// TIA Portal V18 export
// export: Created 2025-12-01T12:39:34.8419056Z, ExportSetting None, DisplayName Totally Integrated Automation Portal, DisplayVersion V18 Update 5, DisplayName TIA Portal Openness, DisplayVersion V18 Update 5, DisplayName TIA Portal Teamcenter Gateway, DisplayVersion V18, DisplayName TIA Portal Version Control Interface, DisplayVersion V18, DisplayName STEP 7 Professional, DisplayVersion V18 Update 5, DisplayName STEP 7 Safety, DisplayVersion V18, DisplayName WinCC Professional, DisplayVersion V18 Update 5
VAR_GLOBAL   // PLC tag table "PLCIO_DQ"
   oHMIControlOn AT %Q100.0 : Bool;   // HMI_上电按钮
   oHMIMachineStart AT %Q100.1 : Bool;   // HMI_设备启动按钮
   oHMIMachineStop AT %Q100.2 : Bool;   // HMI_设备停止按钮
   oHMIResetButton AT %Q100.3 : Bool;   // HMI_复位按钮
   oHMISafetyGateUnlock AT %Q100.4 : Bool;   // HMI_安全门解锁按钮
   "RESERVE_Q100.5" AT %Q100.5 : Bool;   // 备用_Q100.5
   "RESERVE_Q100.6" AT %Q100.6 : Bool;   // 备用_Q100.6
   "RESERVE_Q100.7" AT %Q100.7 : Bool;   // 备用_Q100.7
   "oTowerLight-Green" AT %Q101.0 : Bool;   // 稳光-绿
   "oTowerLight-Red" AT %Q101.1 : Bool;   // 稳光-红
   "oTowerLight-yellow" AT %Q101.2 : Bool;   // 稳光-黄
   "oTowerLight-Blue" AT %Q101.3 : Bool;   // 稳光-蓝
   "oTowerLight-Buzzer" AT %Q101.4 : Bool;   // 蜂鸣
   oLED_lamp_1 AT %Q101.5 : Bool;   // 日光灯_1
   oLED_lamp_2 AT %Q101.6 : Bool;   // 日光灯_2
   oSafetyPLC AT %Q101.7 : Bool;   // 安全PLC
   oSafetyDoorLocked_1 AT %Q102.0 : Bool;   // 安全门锁定_1
   oSafetyDoorLocked_2 AT %Q102.1 : Bool;   // 安全门锁定_2
   oSafetyDoorLocked_3 AT %Q102.2 : Bool;   // 安全门锁定_3
   oSafetyDoorLocked_4 AT %Q102.3 : Bool;   // 安全门锁定_4
   oSafetyDoorLocked_5 AT %Q102.4 : Bool;   // 安全门锁定_5
   oSafetyDoorLocked_6 AT %Q102.5 : Bool;   // 安全门锁定_6
   oSafetyDoorLocked_7 AT %Q102.6 : Bool;   // 安全门锁定_7
   oSafetyDoorLocked_8 AT %Q102.7 : Bool;   // 安全门锁定_8
   oSafetyDoorLocked AT %Q103.0 : Bool;   // 连锁安全门锁定
   "oE-NG-01SafetyGate" AT %Q103.1 : Bool;   // E-NG料盒-01安全门锁
   oMaterielDoorLocked_H2 AT %Q103.4 : Bool;   // 物料门锁定_2
   oMaterielDoorLocked_J1 AT %Q103.5 : Bool;   // 物料门锁定_3
   "oE-NG-02SafetyGate" AT %Q103.2 : Bool;   // E-NG料盒-02安全门锁
   oMaterielDoorLocked_H1 AT %Q103.3 : Bool;   // 物料门锁定_1
   oMaterielDoorLocked_J2 AT %Q103.6 : Bool;   // 物料门锁定_4
   oMaterielDoorLocked_K1 AT %Q103.7 : Bool;   // 物料门锁定_5
   oNG_Button1 AT %Q104.0 : Bool;   // NG下料按钮1
   oNG_Button2 AT %Q104.1 : Bool;   // NG下料按钮2
   oShaft_Button AT %Q104.2 : Bool;   // shaft 上料按钮
   oShaft_EmptyButton AT %Q104.3 : Bool;   // shaft 取空料盘按钮
   oMagnet_Button AT %Q104.4 : Bool;   // Magnet上料按钮
   oMagnet_EmptyButton AT %Q104.5 : Bool;   // Magnet取空料盘按钮
   oMagnet_UnlockButton AT %Q104.6 : Bool;   // Magne门解锁按钮
   "RESERVE_Q104.7" AT %Q104.7 : Bool;   // 备用_Q104.7
   oUnloading_EmptyButton AT %Q105.4 : Bool;   // Unloading取空料盘按钮
   oUnloading_UnlockButton AT %Q105.5 : Bool;   // Unloading门解锁按钮
   oMaterielDoorLocked_K2 AT %Q105.6 : Bool;   // 物料门锁定_6
   oMaterielDoorLocked_L1 AT %Q105.7 : Bool;   // 物料门锁定_7
   oReserved_Button AT %Q105.0 : Bool;   // Reserved上料按钮
   oReserved_EmptyButton AT %Q105.1 : Bool;   // Reserved取空料盘按钮
   oReserved_UnlockButton AT %Q105.2 : Bool;   // Reserved门解锁按钮
   oUnloading_Button AT %Q105.3 : Bool;   // Unloading按钮
   "oC-GluingPro_X" AT %Q106.0 : Bool;   // C-涂胶模组点胶阀_a / C-涂胶系统程序X
   "oC-GluingPro_Y" AT %Q106.1 : Bool;   // C-涂胶模组点胶阀_b / C-涂胶系统程序Y
   "oC-GluingReset" AT %Q106.2 : Bool;   // C-涂胶模组点胶阀_c / C-涂胶系统复位
   "oC-GluingPro_Z" AT %Q106.3 : Bool;   // 备用_Q106.3 / C-涂胶系统程序Z
   "oH-shaftLifting_SpeedChange" AT %Q106.4 : Bool;   // H-shaft 顶升位驱动电机_速度切换
   "oH-shaftLifting_Start" AT %Q106.5 : Bool;   // H-shaft 顶升位驱动电机_启动进料
   "oJ-magnetLifting_SpeedChange" AT %Q106.6 : Bool;   // J-magnet顶升驱动电机_速度切换
   "oJ-magnetLifting_Start" AT %Q106.7 : Bool;   // J-magnet顶升驱动电机_启动进料
   "oK-Lifting3_SpeedChange" AT %Q107.0 : Bool;   // K-预留顶升位3驱动电机_速度切换
   "oK-Lifting3_Start" AT %Q107.1 : Bool;   // K-预留顶升位3驱动电机_启动进料
   "oL-Unloading_CCW" AT %Q107.2 : Bool;   // L-下料线体移栽电机_出料
   "oL-Unloading_CW" AT %Q107.3 : Bool;   // L-下料线体移栽电机_进料
   "oH-shaftLifting_CCWStart" AT %Q107.4 : Bool;   // H-shaft 顶升位驱动电机_启动反转出料
   "oJ-magnetLifting_CCWStart" AT %Q107.5 : Bool;   // J-magnet顶升驱动电机_启动反转出料
   "oK-Lifting3_CCWStart" AT %Q107.6 : Bool;   // K-预留顶升位3驱动电机_启动反转出料
   "RESERVE_Q107.7" AT %Q107.7 : Bool;   // 备用_Q107.7
   "oH-shaftLoading_CCW" AT %Q108.0 : Bool;   // H-shaft上料线体驱动电机_反转
   "oH-shaftLoading_CW" AT %Q108.1 : Bool;   // H-shaft上料线体驱动电机_正转
   "oH-shaftTake_CW" AT %Q108.2 : Bool;   // H-shaft取空盘驱动电机_正转
   "oH-shaftTake_CCW" AT %Q108.3 : Bool;   // H-shaft取空盘驱动电机_反转
   "RESERVE_Q108.4" AT %Q108.4 : Bool;   // 备用_Q108.4
   "RESERVE_Q108.5" AT %Q108.5 : Bool;   // 备用_Q108.5
   "RESERVE_Q108.6" AT %Q108.6 : Bool;   // 备用_Q108.6
   "RESERVE_Q108.7" AT %Q108.7 : Bool;   // 备用_Q108.7
   "RESERVE_Q109.0" AT %Q109.0 : Bool;
   "RESERVE_Q109.1" AT %Q109.1 : Bool;
   "RESERVE_Q109.2" AT %Q109.2 : Bool;
   "RESERVE_Q109.3" AT %Q109.3 : Bool;
   "RESERVE_Q109.4" AT %Q109.4 : Bool;
   "RESERVE_Q109.5" AT %Q109.5 : Bool;
   "RESERVE_Q109.6" AT %Q109.6 : Bool;
   "RESERVE_Q109.7" AT %Q109.7 : Bool;
   "J-magnet Loading _CCW" AT %Q110.0 : Bool;   // J-magnet上料线体驱动电机_反转
   "J-magnet Loading _CW" AT %Q110.1 : Bool;   // J-magnet上料线体驱动电机_正转
   "J-magnet Take _CW" AT %Q110.2 : Bool;   // J-magnet取空盘驱动电机_正转
   "J-magnet Take _CCW" AT %Q110.3 : Bool;   // J-magnet取空盘驱动电机_反转
   "RESERVE_Q110.4" AT %Q110.4 : Bool;   // 备用_Q110.4
   "RESERVE_Q110.5" AT %Q110.5 : Bool;   // 备用_Q110.5
   "RESERVE_Q110.6" AT %Q110.6 : Bool;   // 备用_Q110.6
   "RESERVE_Q110.7" AT %Q110.7 : Bool;   // 备用_Q110.7
   "RESERVE_Q111.0" AT %Q111.0 : Bool;
   "RESERVE_Q111.1" AT %Q111.1 : Bool;
   "RESERVE_Q111.2" AT %Q111.2 : Bool;
   "RESERVE_Q111.3" AT %Q111.3 : Bool;
   "RESERVE_Q111.4" AT %Q111.4 : Bool;
   "RESERVE_Q111.5" AT %Q111.5 : Bool;
   "RESERVE_Q111.6" AT %Q111.6 : Bool;
   "RESERVE_Q111.7" AT %Q111.7 : Bool;
   "L-Unloading _LineMotor_CCW" AT %Q112.0 : Bool;   // K-预留上料线体驱动电机_反转 / L-下料线体驱动电机_反转
   "L-Unloading _LineMotor_CW" AT %Q112.1 : Bool;   // K-预留上料线体驱动电机_正转 / L-下料线体驱动电机_正传
   "K-Take _CW" AT %Q112.2 : Bool;   // K-预留取空盘驱动电机_正转
   "K-Take _CCW" AT %Q112.3 : Bool;   // K-预留取空盘驱动电机_反转
   "RESERVE_Q112.4" AT %Q112.4 : Bool;   // 备用_Q112.4
   "RESERVE_Q112.5" AT %Q112.5 : Bool;   // 备用_Q112.5
   "RESERVE_Q112.6" AT %Q112.6 : Bool;   // 备用_Q112.6
   "RESERVE_Q112.7" AT %Q112.7 : Bool;   // 备用_Q112.7
   "RESERVE_Q113.0" AT %Q113.0 : Bool;
   "RESERVE_Q113.1" AT %Q113.1 : Bool;
   "RESERVE_Q113.2" AT %Q113.2 : Bool;
   "RESERVE_Q113.3" AT %Q113.3 : Bool;
   "RESERVE_Q113.4" AT %Q113.4 : Bool;
   "RESERVE_Q113.5" AT %Q113.5 : Bool;
   "RESERVE_Q113.6" AT %Q113.6 : Bool;
   "RESERVE_Q113.7" AT %Q113.7 : Bool;
   "K-Loading _CCW" AT %Q114.0 : Bool;   // L-下料线体驱动电机_反转 / K-预留上料线体驱动电机_反转
   "K-Loading _CW" AT %Q114.1 : Bool;   // L-下料线体驱动电机_正传 / K-预留上料线体驱动电机_正转
   "RESERVE_Q114.2" AT %Q114.2 : Bool;   // 备用_Q114.2
   "RESERVE_Q114.3" AT %Q114.3 : Bool;   // 备用_Q114.3
   "RESERVE_Q114.4" AT %Q114.4 : Bool;   // 备用_Q114.4
   "RESERVE_Q114.5" AT %Q114.5 : Bool;   // 备用_Q114.5
   "RESERVE_Q114.6" AT %Q114.6 : Bool;   // 备用_Q114.6
   "RESERVE_Q114.7" AT %Q114.7 : Bool;   // 备用_Q114.7
   "RESERVE_Q115.0" AT %Q115.0 : Bool;
   "RESERVE_Q115.1" AT %Q115.1 : Bool;
   "RESERVE_Q115.2" AT %Q115.2 : Bool;
   "RESERVE_Q115.3" AT %Q115.3 : Bool;
   "RESERVE_Q115.4" AT %Q115.4 : Bool;
   "RESERVE_Q115.5" AT %Q115.5 : Bool;
   "RESERVE_Q115.6" AT %Q115.6 : Bool;
   "RESERVE_Q115.7" AT %Q115.7 : Bool;
END_VAR
